{attribute 'qualified_only'}
VAR_GLOBAL CONSTANT
	MOVESTATE_INIT :INT:= 1;
	
	MOVESTATE_ENABLE :INT:= 2;
	MOVESTATE_ENABLE_F :INT:= 21;
	
	MOVESTATE_ERROR :INT:=3;
	MOVESTATE_ERROR_F :INT:=31;
	
	MOVESTATE_RESET : INT:=4;
	MOVESTATE_RESET_F : INT:=41;
	
	MOVESTATE_MOVABS : INT:=5;
	MOVESTATE_MOVABS_I :INT:=50;
	MOVESTATE_MOVABS_F :INT:=51;
	
	MOVESTATE_HOME:  INT:=6;
	MOVESTATE_HOME_I:  INT:=60;
	MOVESTATE_HOME_F:  INT:=61;
END_VAR

(* stored: Version 1.1.0.1, ProductVersion 3.1.4024.4
   GVL QrCts: Id {dee5829f-287a-41f2-8963-8c756a2e5028}, ParameterList True *)
